// SIMATIC STEP 7 (V5.x) project RLI3-ProjetLampe
// CPU: CPU 315-2 DP
// station: Matériel
// station: ST1
// station: P_ADR_BUS
// program: Programme S7(1)

SYMBOL_TABLE
"CYCL_EXC"	OB 1	OB 1	// Cycle Execution
END_SYMBOL_TABLE

ORGANIZATION_BLOCK "CYCL_EXC"	// OB 1
VERSION : 0.1
VAR_TEMP
  Default : ARRAY  [1 .. 20 ] OF BYTE ;
END_VAR
BEGIN
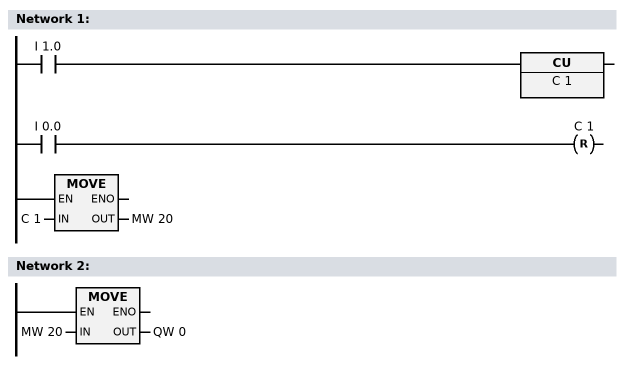
NETWORK
TITLE =
      A     I 1.0;
      CU    C 1;
      NOP   0;
      NOP   0;
      NOP   0;
      A     I 0.0;
      R     C 1;
      L     C 1;
      T     MW 20;
      NOP   0;
      NOP   0;
NETWORK
TITLE =
      L     MW 20;
      T     QW 0;
      NOP   0;
NETWORK
TITLE =
NETWORK
TITLE =
END_ORGANIZATION_BLOCK
